FUNCTION_BLOCK FB_GatoPerro
VAR_INPUT
	RUN 		: BOOL;
END_VAR
VAR_OUTPUT
	Q			: BOOL;
	Gato 		: BOOL;
	Perro 		: BOOL;
	GatoCount 	: UINT;
	PerroCount 	: UINT;

END_VAR
VAR
	R_TRIG_0: R_TRIG;
	R_TRIG_1: R_trig;
	GatoTrigger: BOOL;
	WheelLightTrigger: BOOL;
	R_TRIG_2: R_TRIG;
	RotationTrigger: BOOL;
	RotationCount: UINT;
	ObjectCount: UINT;
	GatoPrime: BOOL;
	bGato_or_Perro: BOOL;
	TON_PrimeDelay: TON;
	WheelTime1: TIME;
	WheelTime3: TIME;
	WheelTime2: TIME;
	GP_Check: UINT;
	//A_RotationMeasure VARs	
		tTimeNow: TIME;
		tRotationTime: TIME;
		tTimeStop: TIME;
		iRotations_In_Minute: DWORD;
		iTimenow: DWORD;
		iOneMinute: DWORD;
		iRotationTime: DWORD;
		iOne_Fourth_Rotations_Time: DWORD;
		iTenth_Of_Rotations_Time: DWORD;
		tOne_Fourth_Rotations_Time: TIME;
		tTenth_Of_Rotations_Time: TIME;
	tonLightSDelay: TON;
	ObjectDetectionTime: TIME := T#50MS;
	Prime_Start: BOOL;
END_VAR

Q := RUN;
A_SensorHandling();

// Rotation counter
IF RotationTrigger THEN
	RotationCount := RotationCount +1;

	// We need slight delay before Priming Gato. Perro could be just nearing the Light sensor and register as Gato
	// Lets calculate rotations per minute, divide it to 3/4th rotation and use these later on to prime Gato just in time
	A_RotationMeasure();
		tRotationTime;			// Informational
		iRotations_In_Minute;	// Informational		
END_IF

// Magnet sensor sees Gato
	// Lets add slight delay to avoid mixing with other object on wheel
	TON_PrimeDelay(IN:= Prime_Start, PT:= tOne_Fourth_Rotations_Time, Q=> , ET=> );
		IF GatoTrigger THEN
			Prime_Start := TRUE;
		END_IF
	// When timer is done, Gato is primed and will register in light sensor
		IF TON_PrimeDelay.Q THEN
			GatoPrime := TRUE;
			Prime_Start := FALSE;
		END_IF

// Light sensor sees an object
IF WheelLightTrigger THEN
	ObjectCount := ObjectCount +1;
	IF NOT GatoPrime THEN			// IF Gato is not primed, its Perro
		PerroCount := PerroCount +1;
		bGato_or_Perro := FALSE;
	ELSE							// If Gato is primed in previous steps, its Gato
		GatoPrime := FALSE;
		GatoCount := GatoCount +1;
		bGato_or_Perro := TRUE;
	END_IF

END_IF

// Which one was it
Gato 	:= bGato_or_Perro;
Perro 	:= NOT bGato_or_Perro;
// Finally, lit up a light for whichever object it was
A_SignalLights();

ACTION A_RotationMeasure:
// Calculate RPM from RotationTime, divide it to 1/4th rotation
// Also 1/10th rotation to filter light sensor input
// If rotation time is slowing too much, or stops, reset to 0.2s


// How long does one rotation take
	tTimeNow := TIME();
	tRotationTime := tTimeNow - tTimeStop;
	tTimeStop := tTimeNow;

//Some conversions:
	iTimenow := TIME_TO_DWORD(tTimeNow);
	iOneMinute := TIME_TO_DWORD(T#1M);
	iRotationTime := TIME_TO_DWORD(tRotationTime);

// Rotations_In_Minute
iRotations_In_Minute :=
	iOneMinute/iRotationTime;
	
// 1/4 and 1/10th rotation times
tOne_Fourth_Rotations_Time := DWORD_TO_TIME( iOne_Fourth_Rotations_Time :=
	iRotationTime/4);
tTenth_Of_Rotations_Time := DWORD_TO_TIME( iTenth_Of_Rotations_Time :=
	iRotationTime/10);
END_ACTION

ACTION A_SensorHandling:
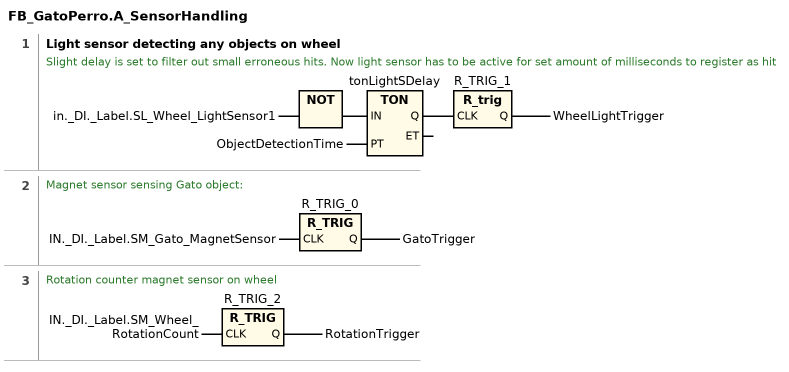
// NETWORK 1: Light sensor detecting any objects on wheel
// Slight delay is set to filter out small erroneous hits. Now light sensor has to be active for set amount of milliseconds to register as hit
tonLightSDelay(IN := NOT in._DI._Label.SL_Wheel_LightSensor1, PT := ObjectDetectionTime); // TON
R_TRIG_1(CLK := tonLightSDelay.Q); // R_trig
WheelLightTrigger := R_TRIG_1.Q;

// NETWORK 2
// Magnet sensor sensing Gato object:
R_TRIG_0(CLK := IN._DI._Label.SM_Gato_MagnetSensor); // R_TRIG
GatoTrigger := R_TRIG_0.Q;

// NETWORK 3
// Rotation counter magnet sensor on wheel
R_TRIG_2(CLK := IN._DI._Label.SM_Wheel_RotationCount); // R_TRIG
RotationTrigger := R_TRIG_2.Q;
END_ACTION

ACTION A_SignalLights:
// Lights signalling which object passed sensor
OUT._DO._Label.LIGHT_White := Gato;
OUT._DO._Label.LIGHT_Green := Perro;
END_ACTION

END_FUNCTION_BLOCK

(* stored: Version 1.1.0.1, ProductVersion 3.1.4024.10
   POU FB_GatoPerro: Id {907c9889-847a-48a2-b378-14a1b7bf9287}, SpecialFunc None
   Action A_RotationMeasure: Id {ed38b022-b882-45b8-9f6c-4ed93bed5869}
   Action A_SensorHandling: Id {9ef9e040-638d-43a8-8a82-3aaf50f53409}
   Action A_SignalLights: Id {3702fc04-dc87-4f5a-8553-8d8da3b39a96} *)
